Staubli VAL3: getZ.pgx

public program getZ(num& nValueZ (dimensions=1))
  local point pHere
begin
  pHere=here(tActive,frActive)
  nValueZ=pHere.trsf.z
end
